Staubli VAL3: CompareTwoPoint.pgx

public program CompareTwoPoint(point x_FirstPoint, point x_SecondPoint, bool& x_bSame)
begin
  //比较两个点是否相同
  x_bSame=false
  if distance(x_FirstPoint,x_SecondPoint)<0.5
    x_bSame=true
  endIf
end
